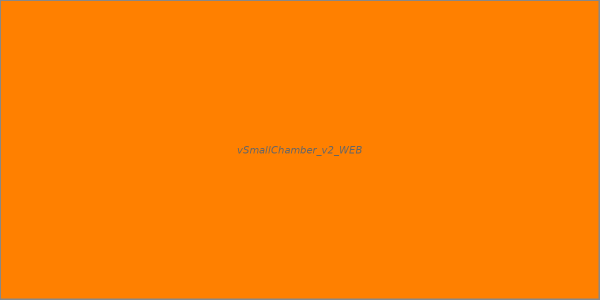
VISUALIZATION vStatusScreen_v2_WEB  // 600x300
VAR_IN_OUT
	arChamber :  fbChamber;
	arParams :    stParamsChamber;
	arControl :    stControl;
END_VAR
    Frame (0,0 600x300)
        shows vSmallChamber_v2_WEB(stParams := arParams, fbChamber := arChamber, stControl := arControl)
END_VISUALIZATION

(* stored: Version 1.1.0.1, ProductVersion 3.1.4024.12
   Visu vStatusScreen_v2_WEB: Id {b524e48f-6933-48f1-b97f-92da7106a812} *)
